Fanuc KAREL source: CHECK_NAME.kl

PROGRAM T
%NOLOCKGROUP
VAR
 v0 : STRING[40]
 v1 : INTEGER
BEGIN
 CHECK_NAME(v0, v1)
END T
